// TIA Portal V17 export
// export: Created 2024-09-02T12:50:39.6950517Z, ExportSetting WithDefaults, DisplayName Totally Integrated Automation Portal, DisplayVersion V17, DisplayName TIA Portal Openness, DisplayVersion V17, DisplayName TIA Portal Version Control Interface, DisplayVersion V17, DisplayName STEP 7 Professional, DisplayVersion V17, DisplayName STEP 7 Safety, DisplayVersion V17, DisplayName WinCC Professional, DisplayVersion V17
TYPE "TypeMobyCommand"
// stored: IsFailsafeCompliant false
   STRUCT
      Sequence { S7_SetPoint := 'True'} : "TypeMobySequence";
      DataBuffer { S7_SetPoint := 'True'} : "TypeMobyDataBuffer";
      BigBuffer : UDInt;
   END_STRUCT;
END_TYPE
